FUNCTION_BLOCK L0_InitService (* Basic Function Block Type *)
  (* Standard: 61499-2 *)
  (* Version 0.0, 2014-09-04, EQUEROL, UJI *)
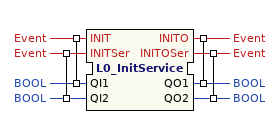
  EVENT_INPUT
    INIT WITH QI1; (* Initialization Request *)
    INITSer WITH QI2; (* Service Initialization completed *)
  END_EVENT
  EVENT_OUTPUT
    INITO WITH QO1; (* Initialization confirmation *)
    INITOSer WITH QO2; (* Service Initialization *)
  END_EVENT
  VAR_INPUT
    QI1 : BOOL; (* Input event qualifier *)
    QI2 : BOOL; (* Input event qualifier *)
  END_VAR
  VAR_OUTPUT
    QO1 : BOOL; (* Output event qualifier *)
    QO2 : BOOL; (* Output event qualifier *)
  END_VAR
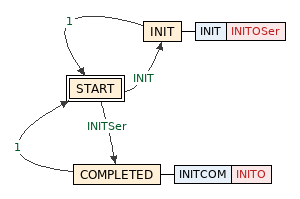
  EC_STATES
    START; (* Initial State *)
    INIT : INIT -> INITOSer; (* Initialization *)
    COMPLETED : INITCOM -> INITO; (* Normal execution *)
  END_STATES
  EC_TRANSITIONS
    START TO INIT := INIT;
    INIT TO START := 1;
    START TO COMPLETED := INITSer;
    COMPLETED TO START := 1;
  END_TRANSITIONS
  ALGORITHM INIT IN ST: (* Initialization algorithm *)
QO2:=QI1;
  END_ALGORITHM
  ALGORITHM INITCOM IN ST: (* Normally executed algorithm *)
QO1:=QI2;
  END_ALGORITHM
END_FUNCTION_BLOCK
